TYPE ST_GundfosMagna3DefaultParameters :
STRUCT
	bExternalTemperatureSensor : BOOL;
END_STRUCT
END_TYPE

(* stored: Version 1.1.0.1, ProductVersion 3.1.4024.9
   DUT ST_GundfosMagna3DefaultParameters: Id {c79135d6-6136-4193-87e6-f0a4d4d2cc36} *)
